(* IEC 61131-3 sources: TheChronoTimer/Portfolio/PLC/Blocks/build, 2 files *)

(* ---- generated_plc.st ---- *)
FUNCTION_BLOCK TFF
  VAR_INPUT
    INPUT : BOOL;
  END_VAR
  VAR
    LATCH : BOOL;
  END_VAR
  VAR_OUTPUT
    OUTPUT : BOOL;
  END_VAR

  LATCH := INPUT;
  OUTPUT := NOT(OUTPUT) AND LATCH OR OUTPUT AND NOT(LATCH);
END_FUNCTION_BLOCK

FUNCTION_BLOCK ONS
  VAR_INPUT
    INPUT : BOOL;
  END_VAR
  VAR_OUTPUT
    OUTPUT : BOOL;
  END_VAR
  VAR
    LATCH : BOOL;
  END_VAR

  OUTPUT := NOT(LATCH) AND INPUT;
  IF INPUT THEN
    LATCH := TRUE; (*set*)
  END_IF;
  IF NOT(INPUT) THEN
    LATCH := FALSE; (*reset*)
  END_IF;
END_FUNCTION_BLOCK

PROGRAM Blocks
  VAR
    INPUT : BOOL;
    OUTPUT0 : BOOL;
    OUTPUT1 : BOOL;
    TFF0 : TFF;
    ONS0 : ONS;
  END_VAR

  TFF0(INPUT := INPUT);
  OUTPUT0 := TFF0.OUTPUT;
  ONS0(INPUT := INPUT);
  OUTPUT1 := ONS0.OUTPUT;
END_PROGRAM

CONFIGURATION Config0

  RESOURCE Res0 ON PLC
    TASK task0(INTERVAL := T#20ms,PRIORITY := 0);
    PROGRAM instance0 WITH task0 : Blocks;
  END_RESOURCE
END_CONFIGURATION

(* ---- plc.st ---- *)
TYPE
  LOGLEVEL : (CRITICAL, WARNING, INFO, DEBUG) := INFO;
END_TYPE

FUNCTION_BLOCK LOGGER
  VAR_INPUT
    TRIG : BOOL;
    MSG : STRING;
    LEVEL : LOGLEVEL := INFO;
  END_VAR
  VAR
    TRIG0 : BOOL;
  END_VAR

  IF TRIG AND NOT TRIG0 THEN
  {{
   LogMessage(GetFbVar(LEVEL),(char*)GetFbVar(MSG, .body),GetFbVar(MSG, .len));
  }}
  END_IF;
  TRIG0:=TRIG;
END_FUNCTION_BLOCK

FUNCTION_BLOCK TFF
  VAR_INPUT
    INPUT : BOOL;
  END_VAR
  VAR
    LATCH : BOOL;
  END_VAR
  VAR_OUTPUT
    OUTPUT : BOOL;
  END_VAR

  LATCH := INPUT;
  OUTPUT := NOT(OUTPUT) AND LATCH OR OUTPUT AND NOT(LATCH);
END_FUNCTION_BLOCK

FUNCTION_BLOCK ONS
  VAR_INPUT
    INPUT : BOOL;
  END_VAR
  VAR_OUTPUT
    OUTPUT : BOOL;
  END_VAR
  VAR
    LATCH : BOOL;
  END_VAR

  OUTPUT := NOT(LATCH) AND INPUT;
  IF INPUT THEN
    LATCH := TRUE; (*set*)
  END_IF;
  IF NOT(INPUT) THEN
    LATCH := FALSE; (*reset*)
  END_IF;
END_FUNCTION_BLOCK

PROGRAM Blocks
  VAR
    INPUT : BOOL;
    OUTPUT0 : BOOL;
    OUTPUT1 : BOOL;
    TFF0 : TFF;
    ONS0 : ONS;
  END_VAR

  TFF0(INPUT := INPUT);
  OUTPUT0 := TFF0.OUTPUT;
  ONS0(INPUT := INPUT);
  OUTPUT1 := ONS0.OUTPUT;
END_PROGRAM

CONFIGURATION Config0

  RESOURCE Res0 ON PLC
    TASK task0(INTERVAL := T#20ms,PRIORITY := 0);
    PROGRAM instance0 WITH task0 : Blocks;
  END_RESOURCE
END_CONFIGURATION
